# EPICS substitutions: roles/install_ioc/tasks/device_types/base_soft_ioc/examples/base-soft-ioc-01/test.substitutions
file "$(TOP)/db/test.db"
{
pattern
{ P		        , R	}
{ "TEST"	, "{PRM:CONFIG}" }
}
